// TIA Portal V20 export
// export: Created 2025-12-01T14:56:58.7691942Z, ExportSetting None, DisplayName Totally Integrated Automation Portal, DisplayVersion V20 Update 3, DisplayName TIA Portal Openness, DisplayVersion V20 Update 3, DisplayName TIA Portal Version Control Interface, DisplayVersion V20 Update 3, DisplayName STEP 7 Professional, DisplayVersion V20 Update 3, DisplayName STEP 7 Safety, DisplayVersion V20 Update 2, DisplayName WinCC Basic/Comfort/Advanced, DisplayVersion V20 Update 3, DisplayName WinCC Professional, DisplayVersion V20 Update 3, DisplayName WinCC Unified, DisplayVersion V20 Update 3
FUNCTION_BLOCK "FB88_GALIBO_HuecoTaco_EnRodillos"   // FB88, LAD
TITLE = Galibo de 5 Alturas (2023)
{ S7_Optimized_Access := 'FALSE' }
AUTHOR : GALIBO
NAME : 20140101
VERSION : 3.0
// stored: AutoNumber false, SetENOAutomatically false
   VAR_INPUT
      Mesa : UInt;
      NumGalibo : UInt;
      pHs_Hueco : Bool;
      pHs_Patin : Bool;
      Avance_Tx : Bool;
      HabilitarLectura : Bool;
      PermisoLectura : Bool;
      Rearmar_ConMesaLibre : Bool;
      V_FiltroHueco : Int;
      V_FiltroPatin : Int;
      V_InicioDePatin : Int;
      V_LongitudDePatin : Int;
   END_VAR
   VAR_OUTPUT
      Codigo : Word;
      Baliza : Bool;
      ErrorHuecoPatin : Bool;
      FinLectura : Bool;
   END_VAR
   VAR_IN_OUT
      SinopticoGalibo_HuecoPatinNOOK : Bool;
      SinopticoGalibo_Señal : "UDT_HMI_SeñalesGalibo";
      SinopticoGalibo_Codigo : Word;
   END_VAR
   VAR
      Filtro_Hueco : "FB910_CNT_UHS";
      Filtro_Patin : "FB910_CNT_UHS";
      CNT_InicioDePatin : "FB910_CNT_UHS";
      CNT_LongitudDePatin { S7_SetPoint := 'True'} : "FB910_CNT_UHS";
      GAL_ET00 : Bool;
      GAL_ET01 : Bool;
      GAL_ET02 : Bool;
      GAL_ET03 : Bool;
      pHsGalibo_OK { ExternalAccessible := 'False'; ExternalVisible := 'False'; ExternalWritable := 'False'} : Bool;
      LeerPatin : Bool;
      MemoDetectorPatin : Bool;
      Patin_OK : Bool;
      Patin_NOK : Bool;
      LeerHueco : Bool;
      Hueco_OK : Bool;
      Hueco_NOK : Bool;
      CodigoHueco : SInt;
      CodigoTaco : SInt;
      MemoCodigo : Word;
      STAT_Baliza_Galibo : Bool;
   END_VAR
   VAR_TEMP
      EstadoZona : "EstadoZona";
      EstadoVI : "EstadosMesa";
   END_VAR
BEGIN

REGION Network 1: INICIALIZAR - Recoger las Variables de Estado de la Mesa
   // Se recoge - Estado_CBx
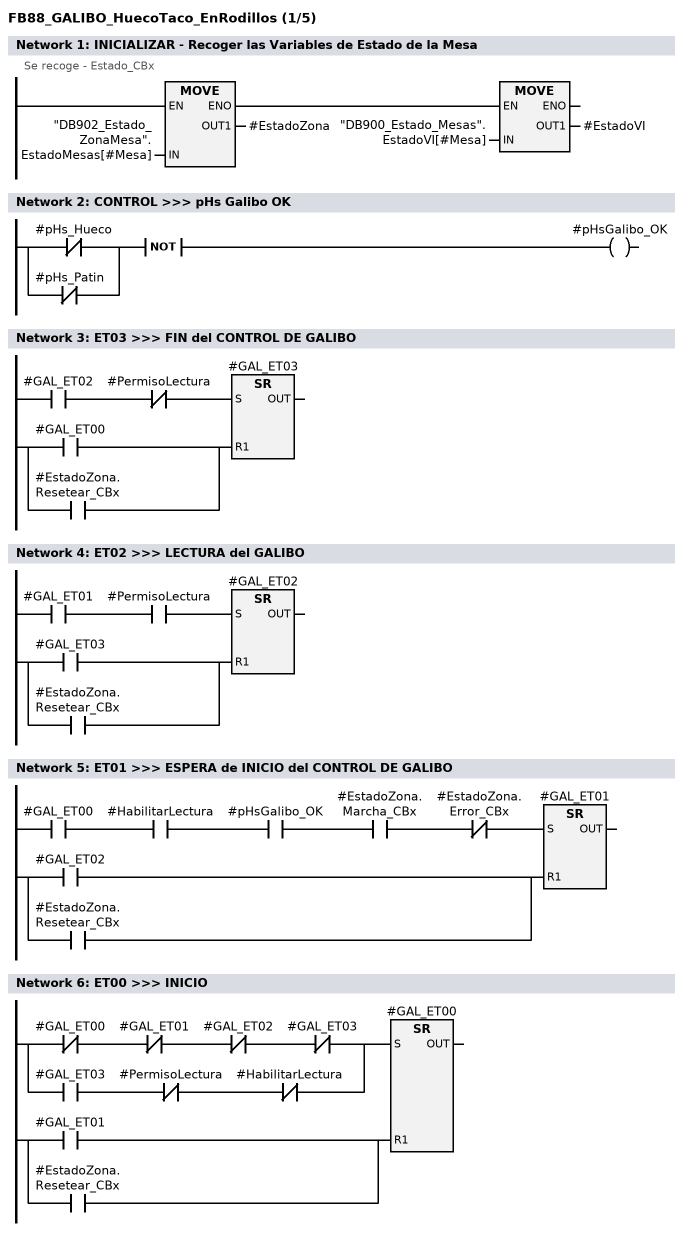
   RUNG wire#powerrail
      Move(in := "DB902_Estado_ZonaMesa".EstadoMesas[#Mesa], out1 => #EstadoZona)
      Move(in := "DB900_Estado_Mesas".EstadoVI[#Mesa], out1 => #EstadoVI)
   END_RUNG
   // the same network as SCL:
   #EstadoZona := "DB902_Estado_ZonaMesa".EstadoMesas[#Mesa];
   #EstadoVI := "DB900_Estado_Mesas".EstadoVI[#Mesa];
END_REGION

REGION Network 2: CONTROL >>> pHs Galibo OK
   RUNG wire#powerrail
      I_Contact( #pHs_Hueco )
      wire#w1
      Not()
      Coil( #pHsGalibo_OK )
   END_RUNG
   RUNG wire#powerrail
      I_Contact( #pHs_Patin )
   END_RUNG wire#w1
   // the same network as SCL:
   #pHsGalibo_OK := NOT (NOT #pHs_Hueco OR NOT #pHs_Patin);
END_REGION

REGION Network 3: ET03 >>> FIN del CONTROL DE GALIBO
   RUNG wire#powerrail
      Contact( #GAL_ET02 )
      I_Contact( #PermisoLectura )
      S_SR(operand := #GAL_ET03, r1 := wire#w1)
   END_RUNG
   RUNG wire#powerrail
      Contact( #GAL_ET00 )
   END_RUNG wire#w1
   RUNG wire#powerrail
      Contact( #EstadoZona.Resetear_CBx )
   END_RUNG wire#w1
   // the same network as SCL:
   IF #GAL_ET02 AND NOT #PermisoLectura THEN
       #GAL_ET03 := TRUE;   // SR flip-flop
   END_IF;
   IF #GAL_ET00 OR #EstadoZona.Resetear_CBx THEN #GAL_ET03 := FALSE; END_IF;
END_REGION

REGION Network 4: ET02 >>> LECTURA del GALIBO
   RUNG wire#powerrail
      Contact( #GAL_ET01 )
      Contact( #PermisoLectura )
      S_SR(operand := #GAL_ET02, r1 := wire#w1)
   END_RUNG
   RUNG wire#powerrail
      Contact( #GAL_ET03 )
   END_RUNG wire#w1
   RUNG wire#powerrail
      Contact( #EstadoZona.Resetear_CBx )
   END_RUNG wire#w1
   // the same network as SCL:
   IF #GAL_ET01 AND #PermisoLectura THEN
       #GAL_ET02 := TRUE;   // SR flip-flop
   END_IF;
   IF #GAL_ET03 OR #EstadoZona.Resetear_CBx THEN #GAL_ET02 := FALSE; END_IF;
END_REGION

REGION Network 5: ET01 >>> ESPERA de INICIO del CONTROL DE GALIBO
   RUNG wire#powerrail
      Contact( #GAL_ET00 )
      Contact( #HabilitarLectura )
      Contact( #pHsGalibo_OK )
      Contact( #EstadoZona.Marcha_CBx )
      I_Contact( #EstadoZona.Error_CBx )
      S_SR(operand := #GAL_ET01, r1 := wire#w1)
   END_RUNG
   RUNG wire#powerrail
      Contact( #GAL_ET02 )
   END_RUNG wire#w1
   RUNG wire#powerrail
      Contact( #EstadoZona.Resetear_CBx )
   END_RUNG wire#w1
   // the same network as SCL:
   IF #GAL_ET00 AND #HabilitarLectura AND #pHsGalibo_OK AND #EstadoZona.Marcha_CBx AND NOT #EstadoZona.Error_CBx THEN
       #GAL_ET01 := TRUE;   // SR flip-flop
   END_IF;
   IF #GAL_ET02 OR #EstadoZona.Resetear_CBx THEN #GAL_ET01 := FALSE; END_IF;
END_REGION

REGION Network 6: ET00 >>> INICIO
   RUNG wire#powerrail
      I_Contact( #GAL_ET00 )
      I_Contact( #GAL_ET01 )
      I_Contact( #GAL_ET02 )
      I_Contact( #GAL_ET03 )
      wire#w1
      S_SR(operand := #GAL_ET00, r1 := wire#w2)
   END_RUNG
   RUNG wire#powerrail
      Contact( #GAL_ET03 )
      I_Contact( #PermisoLectura )
      I_Contact( #HabilitarLectura )
   END_RUNG wire#w1
   RUNG wire#powerrail
      Contact( #GAL_ET01 )
   END_RUNG wire#w2
   RUNG wire#powerrail
      Contact( #EstadoZona.Resetear_CBx )
   END_RUNG wire#w2
   // the same network as SCL:
   IF (NOT #GAL_ET00 AND NOT #GAL_ET01 AND NOT #GAL_ET02 AND NOT #GAL_ET03) OR (#GAL_ET03 AND NOT #PermisoLectura AND NOT #HabilitarLectura) THEN
       #GAL_ET00 := TRUE;   // SR flip-flop
   END_IF;
   IF #GAL_ET01 OR #EstadoZona.Resetear_CBx THEN #GAL_ET00 := FALSE; END_IF;
END_REGION

REGION Network 7: ERROR >>> Fotocelulas de Galibo
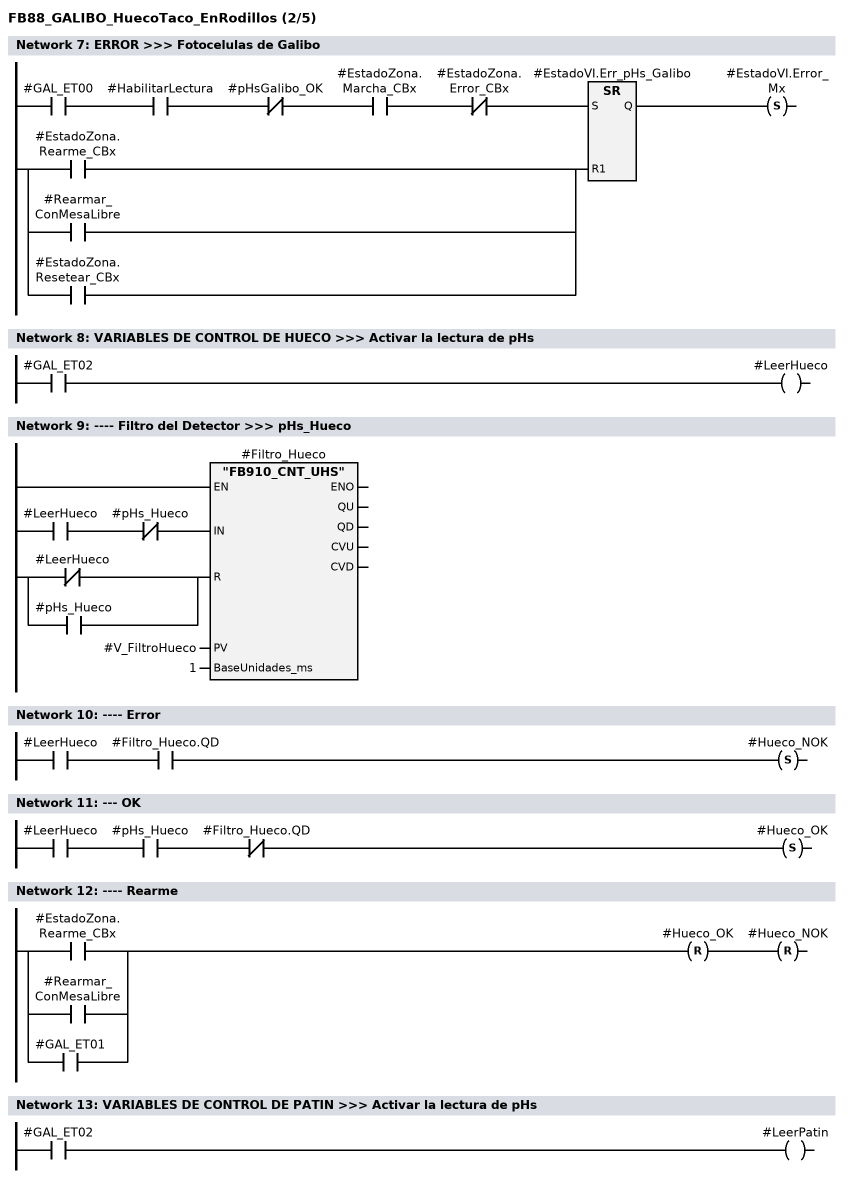
   RUNG wire#powerrail
      Contact( #GAL_ET00 )
      Contact( #HabilitarLectura )
      I_Contact( #pHsGalibo_OK )
      Contact( #EstadoZona.Marcha_CBx )
      I_Contact( #EstadoZona.Error_CBx )
      S_SR(operand := #EstadoVI.Err_pHs_Galibo, r1 := wire#w1)
      S_Coil( #EstadoVI.Error_Mx )
   END_RUNG
   RUNG wire#powerrail
      Contact( #EstadoZona.Rearme_CBx )
   END_RUNG wire#w1
   RUNG wire#powerrail
      Contact( #Rearmar_ConMesaLibre )
   END_RUNG wire#w1
   RUNG wire#powerrail
      Contact( #EstadoZona.Resetear_CBx )
   END_RUNG wire#w1
   // the same network as SCL:
   IF #GAL_ET00 AND #HabilitarLectura AND NOT #pHsGalibo_OK AND #EstadoZona.Marcha_CBx AND NOT #EstadoZona.Error_CBx THEN
       #EstadoVI.Err_pHs_Galibo := TRUE;   // SR flip-flop
   END_IF;
   IF #EstadoZona.Rearme_CBx OR #Rearmar_ConMesaLibre OR #EstadoZona.Resetear_CBx THEN
       #EstadoVI.Err_pHs_Galibo := FALSE;
   END_IF;
   IF #EstadoVI.Err_pHs_Galibo THEN #EstadoVI.Error_Mx := TRUE; END_IF;
END_REGION

REGION Network 8: VARIABLES DE CONTROL DE HUECO >>> Activar la lectura de pHs
   RUNG wire#powerrail
      Contact( #GAL_ET02 )
      Coil( #LeerHueco )
   END_RUNG
   // the same network as SCL:
   #LeerHueco := #GAL_ET02;
END_REGION

REGION Network 9: ---- Filtro del Detector >>> pHs_Hueco
   RUNG wire#powerrail
      #Filtro_Hueco(IN := wire#w1, R := wire#w2, PV := #V_FiltroHueco, BaseUnidades_ms := 1, QU =>, QD =>, CVU =>, CVD =>)
   END_RUNG
   RUNG wire#powerrail
      Contact( #LeerHueco )
      I_Contact( #pHs_Hueco )
   END_RUNG wire#w1
   RUNG wire#powerrail
      I_Contact( #LeerHueco )
   END_RUNG wire#w2
   RUNG wire#powerrail
      Contact( #pHs_Hueco )
   END_RUNG wire#w2
   // the same network as SCL:
   #Filtro_Hueco(IN := #LeerHueco AND NOT #pHs_Hueco,   // "FB910_CNT_UHS"
                 R := NOT #LeerHueco OR #pHs_Hueco,
                 PV := #V_FiltroHueco,
                 BaseUnidades_ms := 1);
END_REGION

REGION Network 10: ---- Error
   RUNG wire#powerrail
      Contact( #LeerHueco )
      Contact( #Filtro_Hueco.QD )
      S_Coil( #Hueco_NOK )
   END_RUNG
   // the same network as SCL:
   IF #LeerHueco AND #Filtro_Hueco.QD THEN #Hueco_NOK := TRUE; END_IF;
END_REGION

REGION Network 11: --- OK
   RUNG wire#powerrail
      Contact( #LeerHueco )
      Contact( #pHs_Hueco )
      I_Contact( #Filtro_Hueco.QD )
      S_Coil( #Hueco_OK )
   END_RUNG
   // the same network as SCL:
   IF #LeerHueco AND #pHs_Hueco AND NOT #Filtro_Hueco.QD THEN #Hueco_OK := TRUE; END_IF;
END_REGION

REGION Network 12: ---- Rearme
   RUNG wire#powerrail
      Contact( #EstadoZona.Rearme_CBx )
      wire#w1
      R_Coil( #Hueco_OK )
      R_Coil( #Hueco_NOK )
   END_RUNG
   RUNG wire#powerrail
      Contact( #Rearmar_ConMesaLibre )
   END_RUNG wire#w1
   RUNG wire#powerrail
      Contact( #GAL_ET01 )
   END_RUNG wire#w1
   // the same network as SCL:
   IF #EstadoZona.Rearme_CBx OR #Rearmar_ConMesaLibre OR #GAL_ET01 THEN
       #Hueco_OK := FALSE;
       #Hueco_NOK := FALSE;
   END_IF;
END_REGION

REGION Network 13: VARIABLES DE CONTROL DE PATIN >>> Activar la lectura de pHs
   RUNG wire#powerrail
      Contact( #GAL_ET02 )
      Coil( #LeerPatin )
   END_RUNG
   // the same network as SCL:
   #LeerPatin := #GAL_ET02;
END_REGION

REGION Network 14: ---- Filtro del Detector >>> pHs_Patin
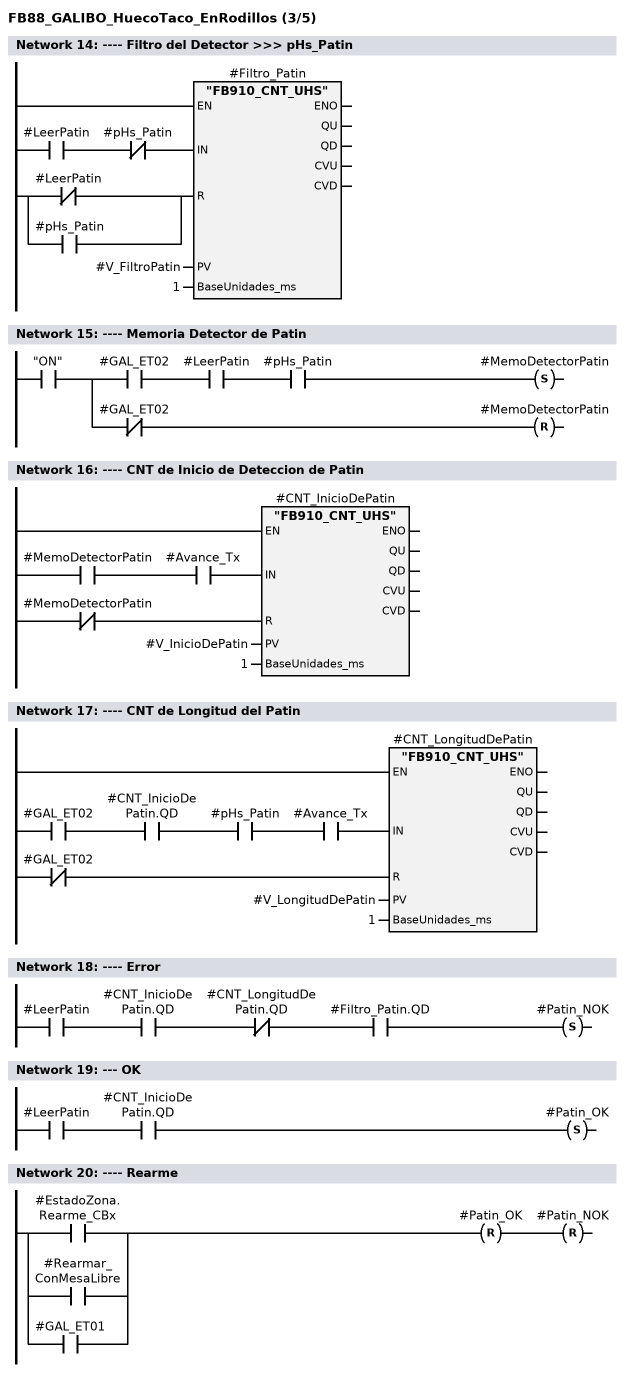
   RUNG wire#powerrail
      #Filtro_Patin(IN := wire#w1, R := wire#w2, PV := #V_FiltroPatin, BaseUnidades_ms := 1, QU =>, QD =>, CVU =>, CVD =>)
   END_RUNG
   RUNG wire#powerrail
      Contact( #LeerPatin )
      I_Contact( #pHs_Patin )
   END_RUNG wire#w1
   RUNG wire#powerrail
      I_Contact( #LeerPatin )
   END_RUNG wire#w2
   RUNG wire#powerrail
      Contact( #pHs_Patin )
   END_RUNG wire#w2
   // the same network as SCL:
   #Filtro_Patin(IN := #LeerPatin AND NOT #pHs_Patin,   // "FB910_CNT_UHS"
                 R := NOT #LeerPatin OR #pHs_Patin,
                 PV := #V_FiltroPatin,
                 BaseUnidades_ms := 1);
END_REGION

REGION Network 15: ---- Memoria Detector de Patin
   RUNG wire#powerrail
      Contact( "ON" )
      wire#w1
      Contact( #GAL_ET02 )
      Contact( #LeerPatin )
      Contact( #pHs_Patin )
      S_Coil( #MemoDetectorPatin )
   END_RUNG
   RUNG wire#w1
      I_Contact( #GAL_ET02 )
      R_Coil( #MemoDetectorPatin )
   END_RUNG
   // the same network as SCL:
   IF "ON" AND #GAL_ET02 AND #LeerPatin AND #pHs_Patin THEN #MemoDetectorPatin := TRUE; END_IF;
   IF "ON" AND NOT #GAL_ET02 THEN #MemoDetectorPatin := FALSE; END_IF;
END_REGION

REGION Network 16: ---- CNT de Inicio de Deteccion de Patin
   RUNG wire#powerrail
      #CNT_InicioDePatin(IN := wire#w1, R := wire#w2, PV := #V_InicioDePatin, BaseUnidades_ms := 1, QU =>, QD =>, CVU =>, CVD =>)
   END_RUNG
   RUNG wire#powerrail
      Contact( #MemoDetectorPatin )
      Contact( #Avance_Tx )
   END_RUNG wire#w1
   RUNG wire#powerrail
      I_Contact( #MemoDetectorPatin )
   END_RUNG wire#w2
   // the same network as SCL:
   #CNT_InicioDePatin(IN := #MemoDetectorPatin AND #Avance_Tx,   // "FB910_CNT_UHS"
                      R := NOT #MemoDetectorPatin,
                      PV := #V_InicioDePatin,
                      BaseUnidades_ms := 1);
END_REGION

REGION Network 17: ---- CNT de Longitud del Patin
   RUNG wire#powerrail
      #CNT_LongitudDePatin(IN := wire#w1, R := wire#w2, PV := #V_LongitudDePatin, BaseUnidades_ms := 1, QU =>, QD =>, CVU =>, CVD =>)
   END_RUNG
   RUNG wire#powerrail
      Contact( #GAL_ET02 )
      Contact( #CNT_InicioDePatin.QD )
      Contact( #pHs_Patin )
      Contact( #Avance_Tx )
   END_RUNG wire#w1
   RUNG wire#powerrail
      I_Contact( #GAL_ET02 )
   END_RUNG wire#w2
   // the same network as SCL:
   #CNT_LongitudDePatin(IN := #GAL_ET02 AND #CNT_InicioDePatin.QD AND #pHs_Patin AND #Avance_Tx,   // "FB910_CNT_UHS"
                        R := NOT #GAL_ET02,
                        PV := #V_LongitudDePatin,
                        BaseUnidades_ms := 1);
END_REGION

REGION Network 18: ---- Error
   RUNG wire#powerrail
      Contact( #LeerPatin )
      Contact( #CNT_InicioDePatin.QD )
      I_Contact( #CNT_LongitudDePatin.QD )
      Contact( #Filtro_Patin.QD )
      S_Coil( #Patin_NOK )
   END_RUNG
   // the same network as SCL:
   IF #LeerPatin AND #CNT_InicioDePatin.QD AND NOT #CNT_LongitudDePatin.QD AND #Filtro_Patin.QD THEN
       #Patin_NOK := TRUE;
   END_IF;
END_REGION

REGION Network 19: --- OK
   RUNG wire#powerrail
      Contact( #LeerPatin )
      Contact( #CNT_InicioDePatin.QD )
      S_Coil( #Patin_OK )
   END_RUNG
   // the same network as SCL:
   IF #LeerPatin AND #CNT_InicioDePatin.QD THEN #Patin_OK := TRUE; END_IF;
END_REGION

REGION Network 20: ---- Rearme
   RUNG wire#powerrail
      Contact( #EstadoZona.Rearme_CBx )
      wire#w1
      R_Coil( #Patin_OK )
      R_Coil( #Patin_NOK )
   END_RUNG
   RUNG wire#powerrail
      Contact( #Rearmar_ConMesaLibre )
   END_RUNG wire#w1
   RUNG wire#powerrail
      Contact( #GAL_ET01 )
   END_RUNG wire#w1
   // the same network as SCL:
   IF #EstadoZona.Rearme_CBx OR #Rearmar_ConMesaLibre OR #GAL_ET01 THEN
       #Patin_OK := FALSE;
       #Patin_NOK := FALSE;
   END_IF;
END_REGION

REGION Network 21: CODIFICACION DEL GALIBO >>> Inicialiar
   // Por Defecto >>> Sin realizar lectura
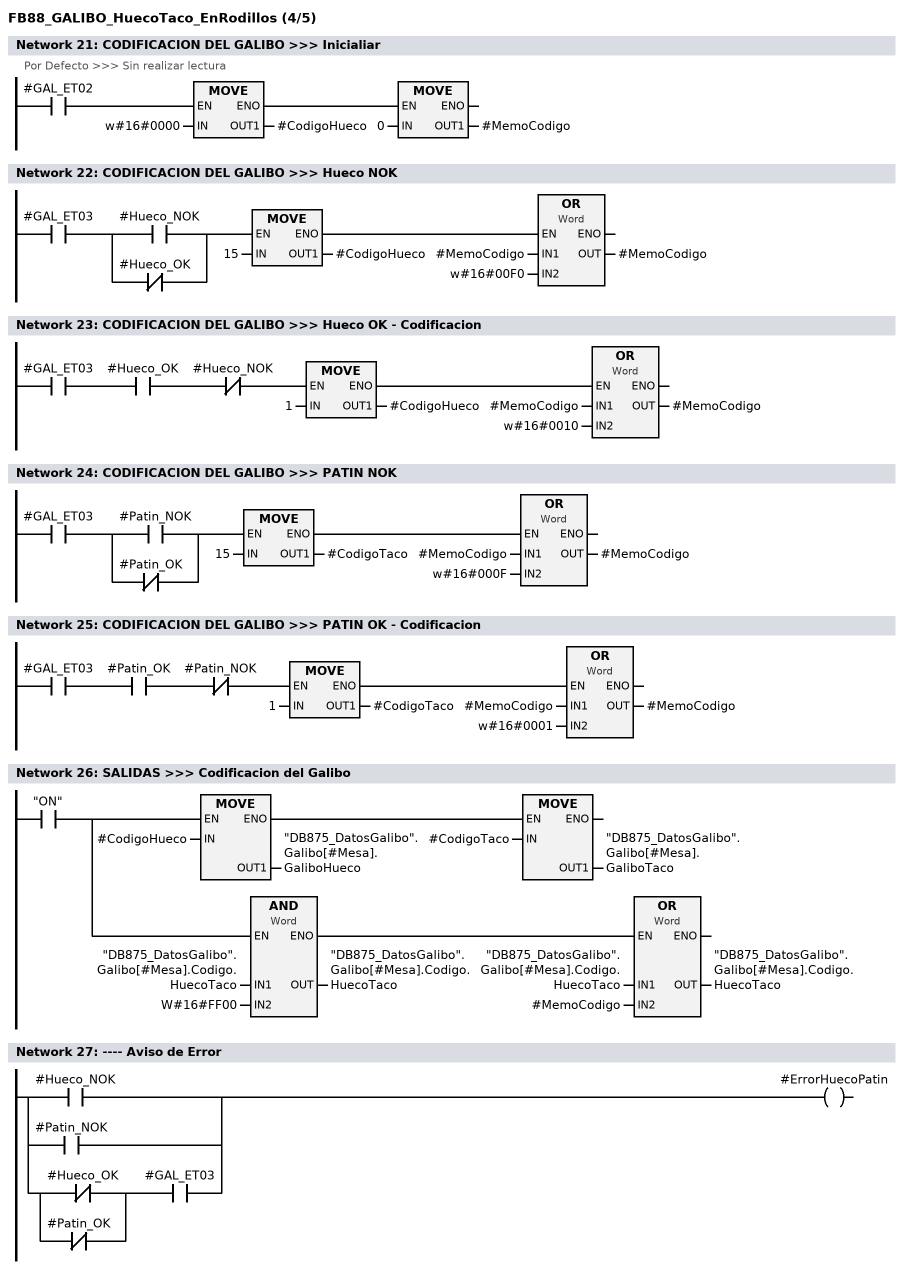
   RUNG wire#powerrail
      Contact( #GAL_ET02 )
      { S7_GenerateENO := "TRUE" } Move(in := w#16#0000, out1 => #CodigoHueco)
      { S7_GenerateENO := "TRUE" } Move(in := 0, out1 => #MemoCodigo)
   END_RUNG
   // the same network as SCL:
   // ENO of a box is taken as its EN; it also drops when the box reports an error
   IF #GAL_ET02 THEN
       #CodigoHueco := w#16#0000;
       #MemoCodigo := 0;
   END_IF;
END_REGION

REGION Network 22: CODIFICACION DEL GALIBO >>> Hueco NOK
   IF #GAL_ET03 AND (#Hueco_NOK OR NOT #Hueco_OK) THEN
       #CodigoHueco := 15;
       #MemoCodigo := #MemoCodigo OR w#16#00F0;
   END_IF;
END_REGION

REGION Network 23: CODIFICACION DEL GALIBO >>> Hueco OK - Codificacion
   IF #GAL_ET03 AND #Hueco_OK AND NOT #Hueco_NOK THEN
       #CodigoHueco := 1;
       #MemoCodigo := #MemoCodigo OR w#16#0010;
   END_IF;
END_REGION

REGION Network 24: CODIFICACION DEL GALIBO >>> PATIN NOK
   IF #GAL_ET03 AND (#Patin_NOK OR NOT #Patin_OK) THEN
       #CodigoTaco := 15;
       #MemoCodigo := #MemoCodigo OR w#16#000F;
   END_IF;
END_REGION

REGION Network 25: CODIFICACION DEL GALIBO >>> PATIN OK - Codificacion
   IF #GAL_ET03 AND #Patin_OK AND NOT #Patin_NOK THEN
       #CodigoTaco := 1;
       #MemoCodigo := #MemoCodigo OR w#16#0001;
   END_IF;
END_REGION

REGION Network 26: SALIDAS >>> Codificacion del Galibo
   // ENO of a box is taken as its EN; it also drops when the box reports an error
   IF "ON" THEN
       "DB875_DatosGalibo".Galibo[#Mesa].GaliboHueco := #CodigoHueco;
       "DB875_DatosGalibo".Galibo[#Mesa].GaliboTaco := #CodigoTaco;
       "DB875_DatosGalibo".Galibo[#Mesa].Codigo.HuecoTaco := "DB875_DatosGalibo".Galibo[#Mesa].Codigo.HuecoTaco AND W#16#FF00;
       "DB875_DatosGalibo".Galibo[#Mesa].Codigo.HuecoTaco := "DB875_DatosGalibo".Galibo[#Mesa].Codigo.HuecoTaco OR #MemoCodigo;
   END_IF;
END_REGION

REGION Network 27: ---- Aviso de Error
   RUNG wire#powerrail
      Contact( #Hueco_NOK )
      wire#w1
      Coil( #ErrorHuecoPatin )
   END_RUNG
   RUNG wire#powerrail
      Contact( #Patin_NOK )
   END_RUNG wire#w1
   RUNG wire#powerrail
      I_Contact( #Hueco_OK )
      wire#w2
      Contact( #GAL_ET03 )
   END_RUNG wire#w1
   RUNG wire#powerrail
      I_Contact( #Patin_OK )
   END_RUNG wire#w2
   // the same network as SCL:
   #ErrorHuecoPatin := #Hueco_NOK OR #Patin_NOK OR ((NOT #Hueco_OK OR NOT #Patin_OK) AND #GAL_ET03);
END_REGION

REGION Network 28: --- Fin de Lectura
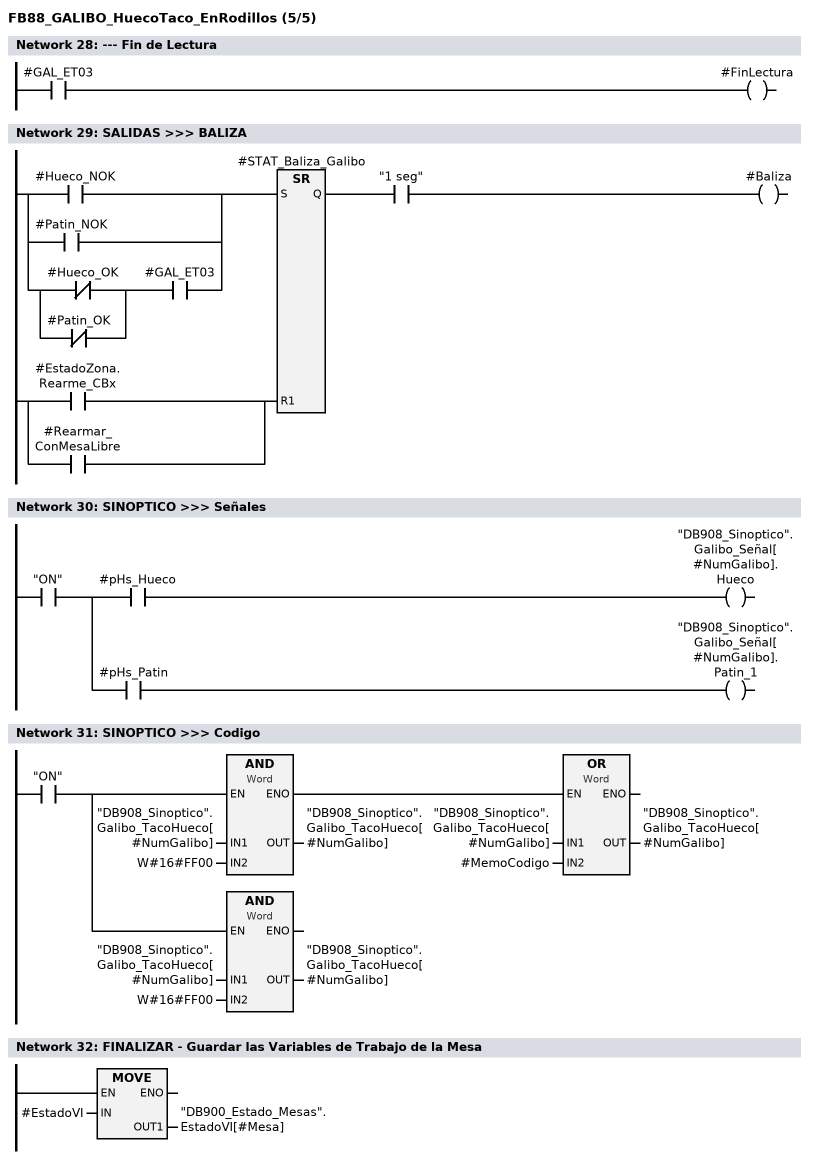
   RUNG wire#powerrail
      Contact( #GAL_ET03 )
      Coil( #FinLectura )
   END_RUNG
   // the same network as SCL:
   #FinLectura := #GAL_ET03;
END_REGION

REGION Network 29: SALIDAS >>> BALIZA
   RUNG wire#powerrail
      Contact( #Hueco_NOK )
      wire#w1
      S_SR(operand := #STAT_Baliza_Galibo, r1 := wire#w3)
      Contact( "1 seg" )
      Coil( #Baliza )
   END_RUNG
   RUNG wire#powerrail
      Contact( #Patin_NOK )
   END_RUNG wire#w1
   RUNG wire#powerrail
      I_Contact( #Hueco_OK )
      wire#w2
      Contact( #GAL_ET03 )
   END_RUNG wire#w1
   RUNG wire#powerrail
      I_Contact( #Patin_OK )
   END_RUNG wire#w2
   RUNG wire#powerrail
      Contact( #EstadoZona.Rearme_CBx )
   END_RUNG wire#w3
   RUNG wire#powerrail
      Contact( #Rearmar_ConMesaLibre )
   END_RUNG wire#w3
   // the same network as SCL:
   IF #Hueco_NOK OR #Patin_NOK OR ((NOT #Hueco_OK OR NOT #Patin_OK) AND #GAL_ET03) THEN
       #STAT_Baliza_Galibo := TRUE;   // SR flip-flop
   END_IF;
   IF #EstadoZona.Rearme_CBx OR #Rearmar_ConMesaLibre THEN #STAT_Baliza_Galibo := FALSE; END_IF;
   #Baliza := #STAT_Baliza_Galibo AND "1 seg";
END_REGION

REGION Network 30: SINOPTICO >>> Señales
   RUNG wire#powerrail
      Contact( "ON" )
      wire#w1
      Contact( #pHs_Hueco )
      Coil( "DB908_Sinoptico".Galibo_Señal[#NumGalibo].Hueco )
   END_RUNG
   RUNG wire#w1
      Contact( #pHs_Patin )
      Coil( "DB908_Sinoptico".Galibo_Señal[#NumGalibo].Patin_1 )
   END_RUNG
   // the same network as SCL:
   "DB908_Sinoptico".Galibo_Señal[#NumGalibo].Hueco := "ON" AND #pHs_Hueco;
   "DB908_Sinoptico".Galibo_Señal[#NumGalibo].Patin_1 := "ON" AND #pHs_Patin;
END_REGION

REGION Network 31: SINOPTICO >>> Codigo
   IF "ON" THEN
       "DB908_Sinoptico".Galibo_TacoHueco[#NumGalibo] := "DB908_Sinoptico".Galibo_TacoHueco[#NumGalibo] AND W#16#FF00;
       "DB908_Sinoptico".Galibo_TacoHueco[#NumGalibo] := "DB908_Sinoptico".Galibo_TacoHueco[#NumGalibo] OR #MemoCodigo;
       "DB908_Sinoptico".Galibo_TacoHueco[#NumGalibo] := "DB908_Sinoptico".Galibo_TacoHueco[#NumGalibo] AND W#16#FF00;
   END_IF;
END_REGION

REGION Network 32: FINALIZAR - Guardar las Variables de Trabajo de la Mesa
   RUNG wire#powerrail
      Move(in := #EstadoVI, out1 => "DB900_Estado_Mesas".EstadoVI[#Mesa])
   END_RUNG
   // the same network as SCL:
   "DB900_Estado_Mesas".EstadoVI[#Mesa] := #EstadoVI;
END_REGION
END_FUNCTION_BLOCK
